// return true if IO is triggerd for a set time period
// only return ture for one cycle, waiting for IO to be released and check for next time
FUNCTION_BLOCK FB_IOToggleCheck
VAR
	// IO type, 0- normally-opend IO; 1- normally-closed IO
	m_IOType :INT :=0;
	
	// counts after IO  is triggerd
	m_IOOnCounts :INT;
	
	// counts threshold indicating IO is trully triggerd
	m_IOOnCountThres :INT :=100;
END_VAR

METHOD check : BOOL
VAR_INPUT
	IOValue :BOOL;
END_VAR
check:=false;
IF (0=m_IOType and IOValue) OR (1=m_IOType AND NOT(IOValue)) THEN
	m_IOOnCounts := MIN(m_IOOnCounts +1, m_IOOnCountThres);
ELSE
	IF m_IOOnCounts>=m_IOOnCountThres THEN
		check:=TRUE;
	END_IF
	 m_IOOnCounts :=0;
END_IF
END_METHOD

METHOD init : BOOL
VAR_INPUT
	i_IOType :INT;
	i_triggerCounts:INT;
END_VAR
m_IOType:=i_IOType;
m_IOOnCountThres := i_triggerCounts;
END_METHOD

END_FUNCTION_BLOCK

(* stored: Version 1.1.0.1, ProductVersion 3.1.4024.11
   POU FB_IOToggleCheck: Id {7ee96876-d402-4755-8a4c-673d3024915f}, SpecialFunc None
   Method check: Id {ddaf28f6-b7c8-41b8-8d5d-b180b564124e}
   Method init: Id {c6e64de0-80ba-4161-8947-1e90294297fc} *)
